// TIA Portal V18 export
TYPE "KukaRobot_UserInput_3"
   STRUCT
      Public : Struct
         GI_TaskMode : USInt;
         GI_PartType : USInt;
         GI_SpeedSet : USInt;
         "GI_PosNo." : USInt;
         GI_5 : Byte;
         GI_6 : Byte;
         GI_7 : Byte;
         GI_8 : Byte;
         GI_9 : Byte;
         GI_10 : Byte;
      END_STRUCT;
      Gripper : Struct
         DI129_Grip1WP : Bool;   // Clamp 1 working position
         DI130_Grip1HP : Bool;   // Clamp 1 original position
         DI131_Grip2WP : Bool;   // Clamp 2 working position
         DI132_Grip2HP : Bool;   // Clamp 2 original position
         DI133_PartOnGrip1 : Bool;   // Is the product Clamp 1 available?
         DI134_PartOnGrip2 : Bool;   // Is there any product for Gripper 2?
         DI135 : Bool;
         DI136 : Bool;
         DI137 : Bool;
         DI138 : Bool;
         DI139 : Bool;
         DI140 : Bool;
         DI141 : Bool;
         DI142 : Bool;
         DI143 : Bool;
         DI144 : Bool;
         DI145 : Bool;
         DI146 : Bool;
         DI147 : Bool;
         DI148 : Bool;
         DI149 : Bool;
         DI150 : Bool;
         DI151 : Bool;
         DI152 : Bool;
         DI153 : Bool;
         DI154 : Bool;
         DI155 : Bool;
         DI156 : Bool;
         DI157 : Bool;
         DI158 : Bool;
         DI159 : Bool;
         DI160 : Bool;
      END_STRUCT;
      Home : Struct
         DI161_HomeSeqStart : Bool;   // The robot can start initialization
         DI162_AutoCycleStart : Bool;   // Robots can start automatic loops
         DI163 : Bool;
         DI164 : Bool;
         DI165 : Bool;
         DI166 : Bool;
         DI167 : Bool;
         DI168 : Bool;
         DI169_RobotMoved : Bool;
         DI170_Robot2_safe_area : Bool;
         DI171 : Bool;
         DI172 : Bool;
         DI173 : Bool;
         DI174 : Bool;
         DI175 : Bool;
         DI176 : Bool;
         DI177_PressNG1_1 : Bool;   // NG1_1 sensor mapping
         DI178_PressNG1_2 : Bool;   // NG1_2 sensor mapping
         DI179_PressNG1_3 : Bool;   // NG1_3 sensor mapping
         DI180_PressNG1_4 : Bool;   // NG1_4 sensor mapping
         DI181_PressNG1_5 : Bool;   // NG1_5 sensor mapping
         DI182_GlueNG2_1 : Bool;   // NG2_1 sensor mapping
         DI183_GlueNG2_2 : Bool;   // NG2_2 sensor mapping
         DI184_GlueNG2_3 : Bool;   // NG2_3 sensor mapping
         DI185_GlueNG2_4 : Bool;   // NG2_4 sensor mapping
         DI186_GlueNG2_5 : Bool;   // NG2_5 sensor mapping
         DI187_ScanNG3_1 : Bool;   // NG3_1 sensor mapping
         DI188_ScanNG3_2 : Bool;   // NG3_2 sensor mapping
         DI189_ScanNG3_3 : Bool;   // NG3_3 sensor mapping
         DI190_ScanNG3_4 : Bool;   // NG3_4 sensor mapping
         DI191_ScanNG3_5 : Bool;   // NG3_5 sensor mapping
         DI192 : Bool;
      END_STRUCT;
      Special : Struct
         DI193 : Bool;
         DI194 : Bool;
         DI195 : Bool;
         DI196 : Bool;
         DI197 : Bool;
         DI198 : Bool;
         DI199 : Bool;
         DI200_Teach_Mode_ON : Bool;
         DI201 : Bool;
         DI202 : Bool;
         DI203 : Bool;
         DI204 : Bool;
         DI205 : Bool;
         DI206 : Bool;
         DI207 : Bool;
         DI208 : Bool;
         DI209 : Bool;
         DI210 : Bool;
         DI211 : Bool;
         DI212 : Bool;
         DI213 : Bool;
         DI214 : Bool;
         DI215 : Bool;
         DI216 : Bool;
         DI217 : Bool;
         DI218 : Bool;
         DI219 : Bool;
         DI220 : Bool;
         DI221 : Bool;
         DI222 : Bool;
         DI223 : Bool;
         DI224 : Bool;
      END_STRUCT;
      Cycle : Struct
         DI225_ScanPosReq : Bool;   // Workwear scan code request
         DI226_ScanPos1Complete : Bool;   // Workwear scan code 1 scan code completed
         DI227_ScanPos2Complete : Bool;   // Workwear scan code 2 scan code completed
         DI228_ScanPos3Complete : Bool;   // Workwear scan code 3 scan code completed
         DI229_ScanPos4Complete : Bool;   // Workwear scan code 4 scan code completed
         DI230_ScanPos5Complete : Bool;   // Workwear scan code 5 scan code completed
         DI231_ScanPos6Complete : Bool;   // Workwear scan code 6 scan code completed
         DI232_ScanPos7Complete : Bool;   // Workwear scan code 7 scan code completed
         DI233 : Bool;
         DI234 : Bool;
         DI235 : Bool;
         DI236 : Bool;
         DI237 : Bool;
         DI238 : Bool;
         DI239 : Bool;
         DI240 : Bool;
         DI241_PickPalletReq : Bool;   // Tray retrieval request
         DI242_NewPallet : Bool;   // New material tray
         DI243 : Bool;
         DI244 : Bool;
         DI245 : Bool;
         DI246 : Bool;
         DI247 : Bool;
         DI248 : Bool;
         DI249_PickMagnetNGReq : Bool;   // Magnet reading code NG picking request
         DI250 : Bool;
         DI251 : Bool;
         DI252 : Bool;
         DI253_PickGlueNGReq : Bool;   // Dispensing NG material retrieval request
         DI254 : Bool;
         DI255 : Bool;
         DI256 : Bool;
         DI257_PickTableReq : Bool;   // Turntable retrieval request
         DI258 : Bool;
         DI259 : Bool;
         DI260 : Bool;
         DI261_ScanRingReq : Bool;   // Ring scan code request
         DI262_ScanRingComplete : Bool;   // Ring scan completed
         DI263 : Bool;
         DI264 : Bool;
         DI265_LoadPressNGReq1 : Bool;   // NG discharge request 1 press-fit NG
         DI266_LoadGlueNGReq2 : Bool;   // NG discharge request 2 Glue NG
         DI267_LoadScanNGReq3 : Bool;   // NG discharge request 3 Scan the code NG
         DI268 : Bool;
         DI269 : Bool;
         DI270 : Bool;
         DI271 : Bool;
         DI272 : Bool;
         DI273_PressPutPart1Req : Bool;
         DI274 : Bool;
         DI275 : Bool;
         DI276 : Bool;
         DI277_PressPutRingReq : Bool;   // Ring jaw 2 press discharge request
         DI278_Press2Leave : Bool;
         DI279 : Bool;
         DI280 : Bool;
         DI281_PressPickPartReq : Bool;   // Press unloading
         DI282 : Bool;
         DI283 : Bool;
         DI284 : Bool;
         DI285 : Bool;
         DI286 : Bool;
         DI287 : Bool;
         DI288 : Bool;
         DI289_PutOkPartReq : Bool;   // Finished parts blanking request
         DI290_UnloadingNewPallet : Bool;   // New pallet for unloading finished parts
         DI291 : Bool;
         DI292 : Bool;
         DI293 : Bool;
         DI294 : Bool;
         DI295 : Bool;
         DI296 : Bool;
         DI297_MaintainRequest : Bool;
         DI298 : Bool;
         DI299 : Bool;
         DI300_HomeRequest : Bool;
         DI301 : Bool;
         DI302 : Bool;
         DI303 : Bool;
         DI304 : Bool;
         DI305_GripScan : Bool;
         DI306_ScanPartComplete : Bool;
         DI307_ScanPartFinish : Bool;
         DI308 : Bool;
         DI309 : Bool;
         DI310 : Bool;
         DI311 : Bool;
         DI312 : Bool;
         DI313 : Bool;
         DI314 : Bool;
         DI315 : Bool;
         DI316 : Bool;
         DI317 : Bool;
         DI318 : Bool;
         DI319 : Bool;
         DI320 : Bool;
         DI321 : Bool;
         DI322 : Bool;
         DI323 : Bool;
         DI324 : Bool;
         DI325 : Bool;
         DI326 : Bool;
         DI327 : Bool;
         DI328 : Bool;
         DI329 : Bool;
         DI330 : Bool;
         DI331 : Bool;
         DI332 : Bool;
         DI333 : Bool;
         DI334 : Bool;
         DI335 : Bool;
         DI336 : Bool;
         Camera_Y : DInt;
         Camera_Z : DInt;
         Camera_R : DInt;
      END_STRUCT;
      Safety : Struct
         DI433 : Bool;
         DI434 : Bool;
         DI435 : Bool;
         DI436 : Bool;
         DI437 : Bool;
         DI438 : Bool;
         DI439 : Bool;
         DI440 : Bool;
         DI441 : Bool;
         DI442 : Bool;
         DI443 : Bool;
         DI444 : Bool;
         DI445 : Bool;
         DI446 : Bool;
         DI447 : Bool;
         DI448 : Bool;
         DI449 : Bool;
         DI450 : Bool;
         DI451 : Bool;
         DI452 : Bool;
         DI453 : Bool;
         DI454 : Bool;
         DI455 : Bool;
         DI456 : Bool;
         DI457 : Bool;
         DI458 : Bool;
         DI459 : Bool;
         DI460 : Bool;
         DI461 : Bool;
         DI462 : Bool;
         DI463 : Bool;
         DI464 : Bool;
         DI465 : Bool;
         DI466 : Bool;
         DI467 : Bool;
         DI468 : Bool;
         DI469 : Bool;
         DI470 : Bool;
         DI471 : Bool;
         DI472 : Bool;
         DI473 : Bool;
         DI474 : Bool;
         DI475 : Bool;
         DI476 : Bool;
         DI477 : Bool;
         DI478 : Bool;
         DI479 : Bool;
         DI480 : Bool;
         DI481 : Bool;
         DI482 : Bool;
         DI483 : Bool;
         DI484 : Bool;
         DI485 : Bool;
         DI486 : Bool;
         DI487 : Bool;
         DI488 : Bool;
         DI489 : Bool;
         DI490 : Bool;
         DI491 : Bool;
         DI492 : Bool;
         DI493 : Bool;
         DI494 : Bool;
         DI495 : Bool;
         DI496 : Bool;
         DI497 : Bool;
         DI498 : Bool;
         DI499 : Bool;
         DI500 : Bool;
         DI501 : Bool;
         DI502 : Bool;
         DI503 : Bool;
         DI504 : Bool;
         DI505 : Bool;
         DI506 : Bool;
         DI507 : Bool;
         DI508 : Bool;
         DI509 : Bool;
         DI510 : Bool;
         DI511 : Bool;
         DI512 : Bool;
      END_STRUCT;
   END_STRUCT;
END_TYPE
